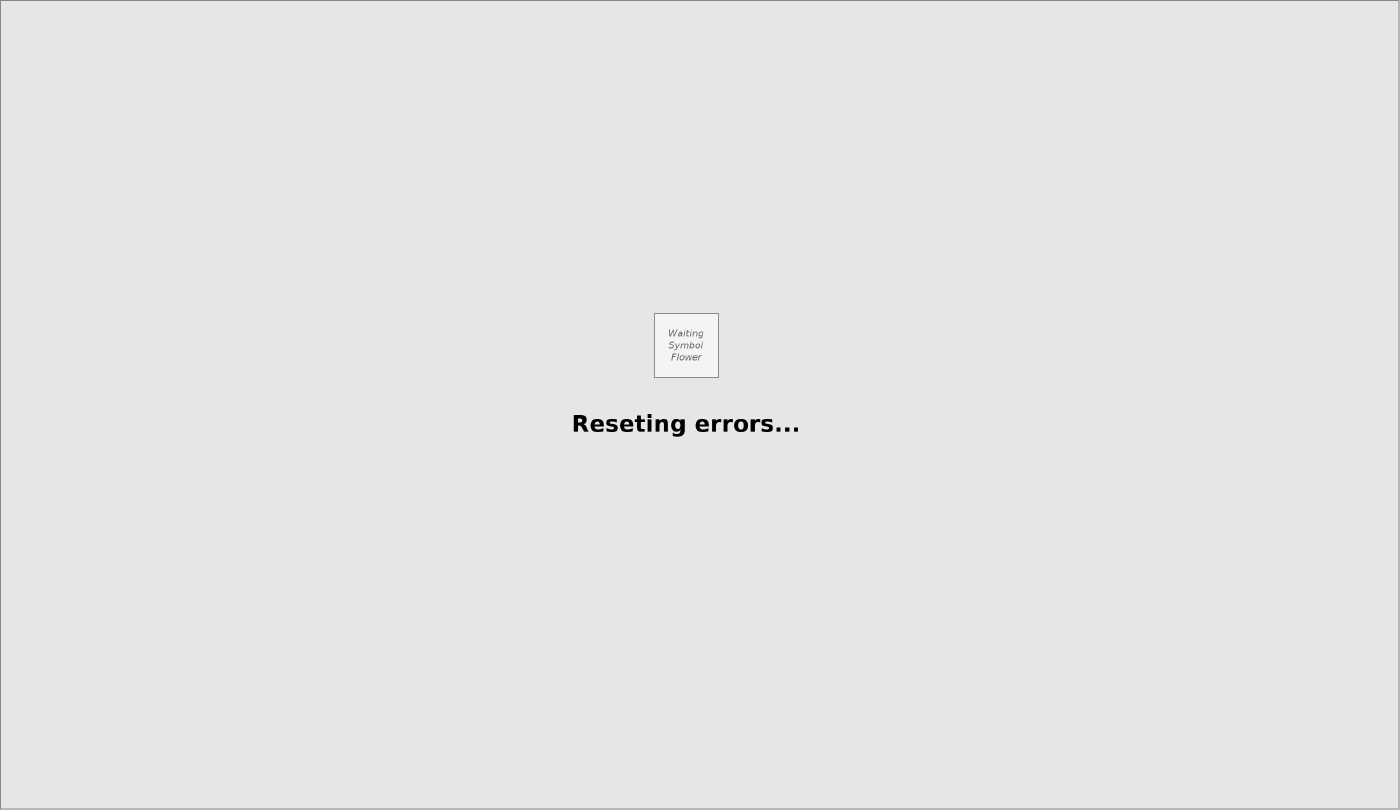
VISUALIZATION PageReset_1  // 1520x880
    WaitingSymbolFlower (710,340 70x70)
    Label (570,440 350x40), "Reseting errors..."
END_VISUALIZATION

(* stored: Version 1.1.0.1, ProductVersion 3.1.4024.12
   Visu PageReset_1: Id {48c979ce-1842-4bb6-a24c-2bb67eeda2dd} *)
